// TIA Portal V17 export
// export: Created 2025-03-07T09:18:46.1410368Z, ExportSetting WithDefaults, DisplayName Totally Integrated Automation Portal, DisplayVersion V17 Update 8, DisplayName TIA Portal Openness, DisplayVersion V17 Update 8, DisplayName TIA Portal Version Control Interface, DisplayVersion V17, DisplayName SINAMICS Startdrive Advanced, DisplayVersion V17 SP2, DisplayName SINAMICS Startdrive G110M, G120, G120C, G120D, G120P, G115D, DisplayVersion V17 SP2, DisplayName SINAMICS Startdrive G130, G150, S120, S150, SINAMICS MV, S210, DisplayVersion V17 SP2, DisplayName STEP 7 Professional, DisplayVersion V17 Update 8, DisplayName SINUMERIK ONE STEP 7 Toolbox, DisplayVersion V17 Update 12, DisplayName SINUMERIK 840D sl STEP 7 Toolbox, DisplayVersion V17 Update 12, DisplayName STEP 7 Safety, DisplayVersion V17 Update 6, DisplayName WinCC Advanced, DisplayVersion V17 Update 8
DATA_BLOCK "DB2391_SAVE_ENERGY"   // DB2391
{ S7_Optimized_Access := 'FALSE'; DB_Accessible_From_OPC_UA := 'FALSE' }
AUTHOR : ETXETAR
VERSION : 1.0
// stored: AutoNumber false, DBAccessibleFromOPCUA false, DBAccessibleFromWebserver true, IsOnlyStoredInLoadMemory false, IsWriteProtectedInAS false
   VAR RETAIN
      SWITCH_OFF_AUX_SERVICES : Bool;   // SAVE ENERGY SWITCH OFF AUXILIARY SERVICES / SWITCH OFF AUXILIARY SERVICES
      SWITCH_OFF_MAIN_SERVICES : Bool;   // SAVE ENERGY SWITCH OFF MAIN SERVICES / SWITCH OFF MAIN SERVICES
      SWITCH_OFF_MAIN_SERVICES_AUX : Bool;   // SAVE ENERGY SWITCH OFF MAIN SERVICES / SWITCH OFF MAIN SERVICES AUXILIARY
      RUN_OUT_REQ : Bool;   // SAVE ENERGY RUNOUT REQUEST / RUN OUT REQUEST
      RESET_TIMERS : Bool;   // SAVE ENERGY RESET TIMERS / RESET TIMERS
      ENABLE_SYSTEM : Bool;   // SAVE ENERGY ENABLE SYSTEM / ENABLE SYSTEM
      HMI_LOW_PRESSURE_DRY_CYCLE : Bool;   // SAVE ENERGY LOW PRESSURE HMI / HMI LOW PRESSURE IN DRY CYCLE
      LOW_PRESSURE_DRY_CYCLE : Bool;   // SAVE ENERGY ENABLE LOW PRESSURE WHILE DRY CYCLE / ENABLE LOW PRESSURE IN DRY CYCLE
      HMI_HIGH_PRESSURE_DRY_CYCLE : Bool;   // SAVE ENERGY HIGH PRESSURE HMI / HMI HIGH PRESSURE IN DRY CYCLE
      HIGH_PRESSURE_DRY_CYCLE : Bool;   // SAVE ENERGY ENABLE HIGH PRESSURE WHILE DRY CYCLE / ENABLE HIGH PRESSURE IN DRY CYCLE
      HMI_FLUSH_PISTOL : Bool;   // SAVE ENERGY FLUSH PISTOL HMI / HMI FLUSH PISTOL
      FLUSH_PISTOL : Bool;   // SAVE ENERGY ENABLE FLUSH PISTOL / ENABLE FLUSH PISTOL
      MINUS_PULSED : Bool;   // SAVE ENERGY MINUS PULSED / MINUS PULSED
      PLUS_PULSED : Bool;   // SAVE ENERGY PLUS PULSED / PLUS PULSED
      SWITCH_OFF_MAIN_SERVICES_MEMORY : Bool;   // SAVE ENERGY SWITCH OFF MAIN SERVICES MEMORY / SWITCH OFF MAIN SERVICES MEMORY
      HMI_MQL_DRY_CYCLE : Bool;   // SAVE ENERGY MQL HMI / HMI MQL IN DRY CYCLE
      MQL_DRY_CYCLE : Bool;   // SAVE ENERGY ENABLE MQL / ENABLE MQL IN DRY CYCLE
      AUX_SERVICES_TIMER_ON : Bool;   // SAVE ENERGY AUXILIARY TIMER ON / AUXILIARY SERVICES TIMER ON
      MAIN_SERVICES_TIMER_ON : Bool;   // SAVE ENERGY MAIN TIMER ON / MAIN SERVICES TIMER ON
      AUX_SERVICES_OFF : Bool;   // SAVE ENERGY AUXILIARY SERVICES OFF / AUXILIARY SERVICES OFF
      MAIN_SERVICES_OFF : Bool;   // SAVE ENERGY MAIN SERVICES OFF / MAIN SERVICES OFF
      TIMER_VALUES_OK : Bool;   // SAVE ENERGY CORRECT TIME DELAY VALUES / TIMER VALUES OK
      AUX_SERVICES_TIME_LEFT : Time;   // AUXILIAR SERVICES TIME MINUTES LEFT / SWITCH OFF AUXILIARY SERVICES TIME LEFT
      MAIN_SERVICES_TIME_LEFT : Time;   // MAIN SERVICES TIME MINUTES LEFT / SWTICH OFF MAIN SERVICES TIME LEFT
      TIMER_RUN_OUT : TON_TIME;   // RUN OUT TIMER
      TIMER_SWITCH_OFF_MAIN_SERVICES : TON_TIME;   // SWITCH OFF MAIN SERVICES TIMER
      TIMER_SWITCH_OFF_AUX_SERVICES : TON_TIME;   // SWITCH OFF AUXILIARY SERVICES TIMER
   END_VAR
BEGIN
   TIMER_RUN_OUT.PT := T#5m;
   TIMER_SWITCH_OFF_MAIN_SERVICES.PT := T#0S;   // SWITCH OFF MAIN SERVICES TIME
   TIMER_SWITCH_OFF_AUX_SERVICES.PT := T#0S;   // SWITCH OFF AUXILIARY SERVICES TIME
END_DATA_BLOCK
